VAR_GLOBAL
// FIO (FactoryIO)
	


	FIO_Input1: ARRAY [0..15] OF BOOL;
	FIO_Input2: ARRAY [0..15] OF BOOL;
	FIO_InputReg: ARRAY [0..7] OF INT;
	FIO_Output1: ARRAY [0..15] OF BOOL;
	FIO_Output2: ARRAY [0..15] OF BOOL;
	FIO_OutputReg: ARRAY [0..7] OF INT;
	
	test: INT;
	
	bOutput1: INT;
END_VAR

(* stored: Version 1.1.0.1, ProductVersion 3.1.4024.11
   GVL GVL_FactoryIO: Id {a4883462-1cb0-43b2-bb87-d6ce56b75e06} *)
